// TIA Portal V20 export
TYPE "LWONIK_typeScrapBoxMonitoring"
// stored: Access Published
   STRUCT
      lock : Bool;
      unlock : Bool;
      reset : Bool;
      error : Bool;
   END_STRUCT;
END_TYPE
